// TIA Portal V16 export
// export: Created 2023-08-28T09:37:47.5616643Z, ExportSetting WithDefaults, DisplayName Totally Integrated Automation Portal, DisplayVersion V16 Update 6, DisplayName TIA Portal Version Control Interface, DisplayVersion V16 Update 2, DisplayName TIA Portal Openness, DisplayVersion V16 Update 6, DisplayName STEP 7 Professional, DisplayVersion V16 Update 6, DisplayName STEP 7 Safety, DisplayVersion V16, DisplayName WinCC Advanced, DisplayVersion V16 Update 6
DATA_BLOCK "MB_SLAVE_RTU_DB"   // DB58
// stored: AutoNumber true, DBAccessibleFromOPCUA true, InstanceOfName MB_SLAVE, OfSystemLibElement MB_SLAVE, OfSystemLibVersion 2.1
"MB_SLAVE"
   // // inherited from MB_BASE
   // VAR
   //    S_PORT : UInt;
   //    S_RESP_TO : UInt;
   //    S_ICHAR_GAP : UInt;
   //    S_RETRIES : UInt;
   // END_VAR
   // VAR_INPUT
   //    MB_ADDR : UInt;
   // END_VAR
   // VAR_OUTPUT
   //    NDR : Bool;
   //    DR : Bool;
   //    ERROR : Bool;
   //    STATUS : Word;
   // END_VAR
   // VAR_IN_OUT
   //    MB_HOLD_REG : Variant;
   // END_VAR
   // VAR
   //    SEND_PTP_SFB : Array[0..11] of Byte;
   //    RCV_PTP_SFB : Array[0..11] of Byte;
   //    MB_State : Word;
   //    Request_Count : Word;
   //    Slave_Message_Count : Word;
   //    Bad_CRC_Count : Word;
   //    Broadcast_Count : Word;
   //    Exception_Count : Word;
   //    Success_Count : Word;
   //    SL_Status_Hold : Word;
   //    HR_Start_Offset : Word;
   //    Init_OK : Bool;
   //    Broadcast_Flag : Bool;
   //    SL_Error_State : Bool;
   //    Extended_Addressing : Bool;
   //    XMT_Set_NDR : Bool;
   //    XMT_Set_DR : Bool;
   // END_VAR
BEGIN
END_DATA_BLOCK
